# EPICS autosave request: iocBoot/iocAMControls/auto_settings.req
file "amControls.req", P=$(P), R=$(R)
file "amControls_settings.req", P=$(P), R=$(R)
